// Mitsubishi GX Developer project: may ghep doc 2   PLC: FX1N

PROGRAM MAIN
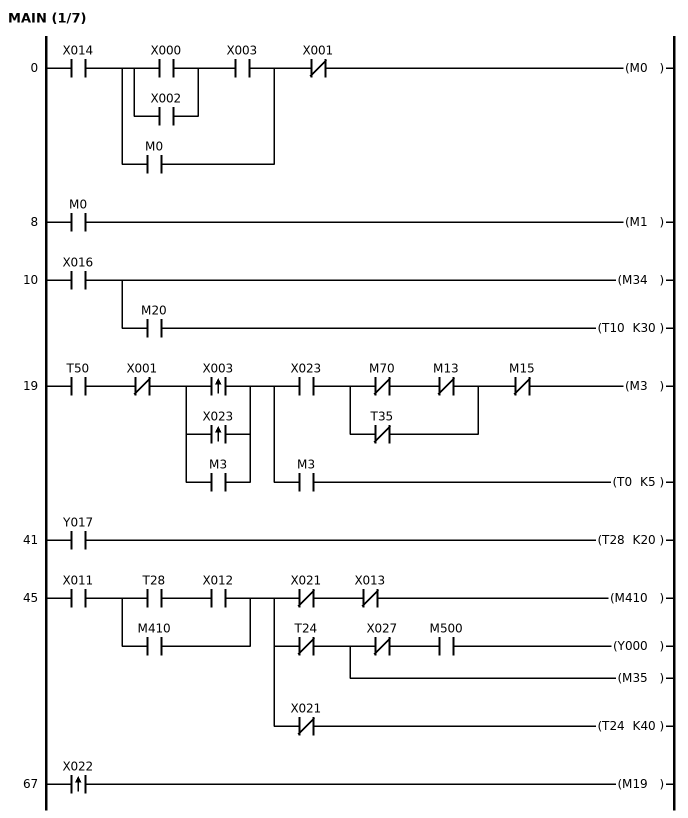
0     LD      X014
      LD      X000
      OR      X002
      AND     X003
      OR      M0
      ANB
      ANI     X001
      OUT     M0
8     LD      M0
      OUT     M1
10    LD      X016
      OUT     M34
      AND     M20
      OUT     T10 K30
19    LD      T50
      ANI     X001
      LDP     X003
      ORP     X023
      OR      M3
      ANB
      MPS
      AND     X023
      LDI     M70
      ANI     M13
      ORI     T35
      ANB
      ANI     M15
      OUT     M3
      MPP
      AND     M3
      OUT     T0 K5
41    LD      Y017
      OUT     T28 K20
45    LD      X011
      LD      T28
      AND     X012
      OR      M410
      ANB
      MPS
      ANI     X021
      ANI     X013
      OUT     M410
      MRD
      ANI     T24
      MPS
      ANI     X027
      AND     M500
      OUT     Y000
      MPP
      OUT     M35
      MPP
      ANI     X021
      OUT     T24 K40
67    LDP     X022
      OUT     M19
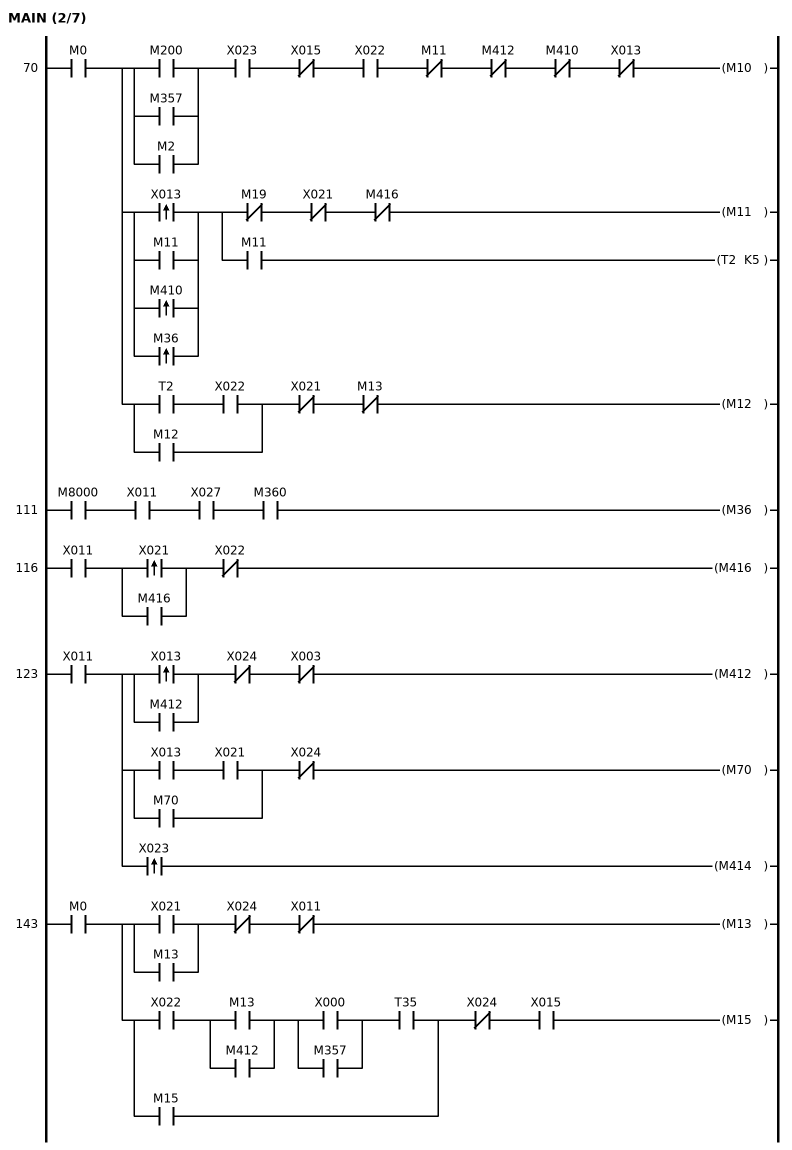
70    LD      M0
      MPS
      LD      M200
      OR      M357
      OR      M2
      ANB
      AND     X023
      ANI     X015
      AND     X022
      ANI     M11
      ANI     M412
      ANI     M410
      ANI     X013
      OUT     M10
      MRD
      LDP     X013
      OR      M11
      ORP     M410
      ORP     M36
      ANB
      MPS
      ANI     M19
      ANI     X021
      ANI     M416
      OUT     M11
      MPP
      AND     M11
      OUT     T2 K5
      MPP
      LD      T2
      AND     X022
      OR      M12
      ANB
      ANI     X021
      ANI     M13
      OUT     M12
111   LD      M8000
      AND     X011
      AND     X027
      AND     M360
      OUT     M36
116   LD      X011
      LDP     X021
      OR      M416
      ANB
      ANI     X022
      OUT     M416
123   LD      X011
      MPS
      LDP     X013
      OR      M412
      ANB
      ANI     X024
      ANI     X003
      OUT     M412
      MRD
      LD      X013
      AND     X021
      OR      M70
      ANB
      ANI     X024
      OUT     M70
      MPP
      ANDP    X023
      OUT     M414
143   LD      M0
      MPS
      LD      X021
      OR      M13
      ANB
      ANI     X024
      ANI     X011
      OUT     M13
      MPP
      LD      X022
      LD      M13
      OR      M412
      ANB
      LD      X000
      OR      M357
      ANB
      AND     T35
      OR      M15
      ANB
      ANI     X024
      AND     X015
      OUT     M15
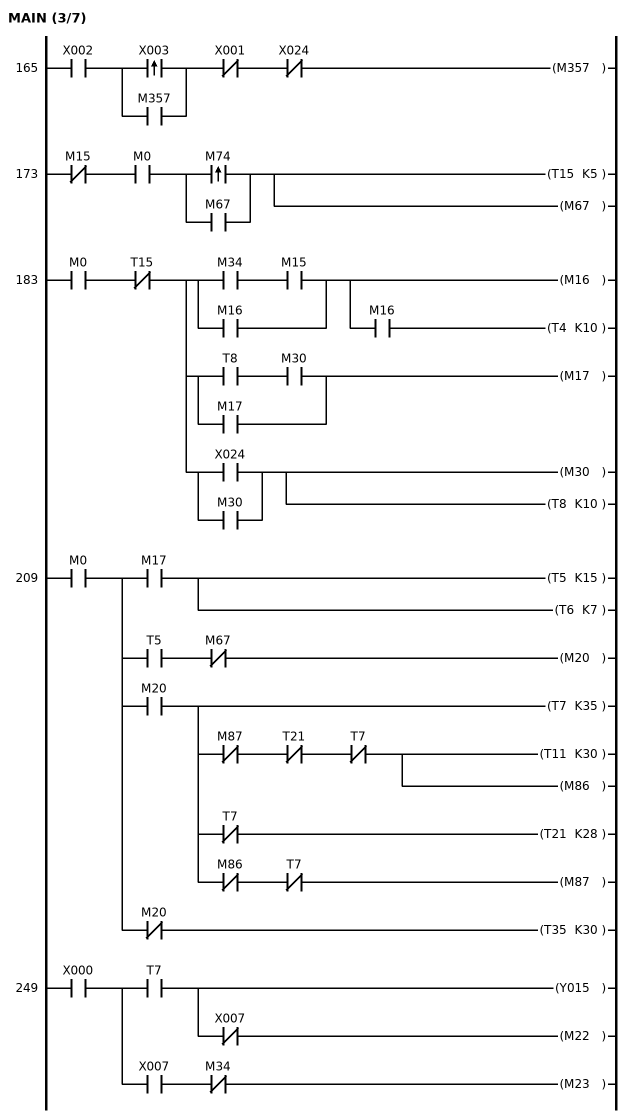
165   LD      X002
      LDP     X003
      OR      M357
      ANB
      ANI     X001
      ANI     X024
      OUT     M357
173   LDI     M15
      AND     M0
      LDP     M74
      OR      M67
      ANB
      OUT     T15 K5
      OUT     M67
183   LD      M0
      ANI     T15
      MPS
      LD      M34
      AND     M15
      OR      M16
      ANB
      OUT     M16
      AND     M16
      OUT     T4 K10
      MRD
      LD      T8
      AND     M30
      OR      M17
      ANB
      OUT     M17
      MPP
      LD      X024
      OR      M30
      ANB
      OUT     M30
      OUT     T8 K10
209   LD      M0
      MPS
      AND     M17
      OUT     T5 K15
      OUT     T6 K7
      MRD
      AND     T5
      ANI     M67
      OUT     M20
      MRD
      AND     M20
      OUT     T7 K35
      MPS
      ANI     M87
      ANI     T21
      ANI     T7
      OUT     T11 K30
      OUT     M86
      MRD
      ANI     T7
      OUT     T21 K28
      MPP
      ANI     M86
      ANI     T7
      OUT     M87
      MPP
      ANI     M20
      OUT     T35 K30
249   LD      X000
      MPS
      AND     T7
      OUT     Y015
      ANI     X007
      OUT     M22
      MPP
      AND     X007
      ANI     M34
      OUT     M23
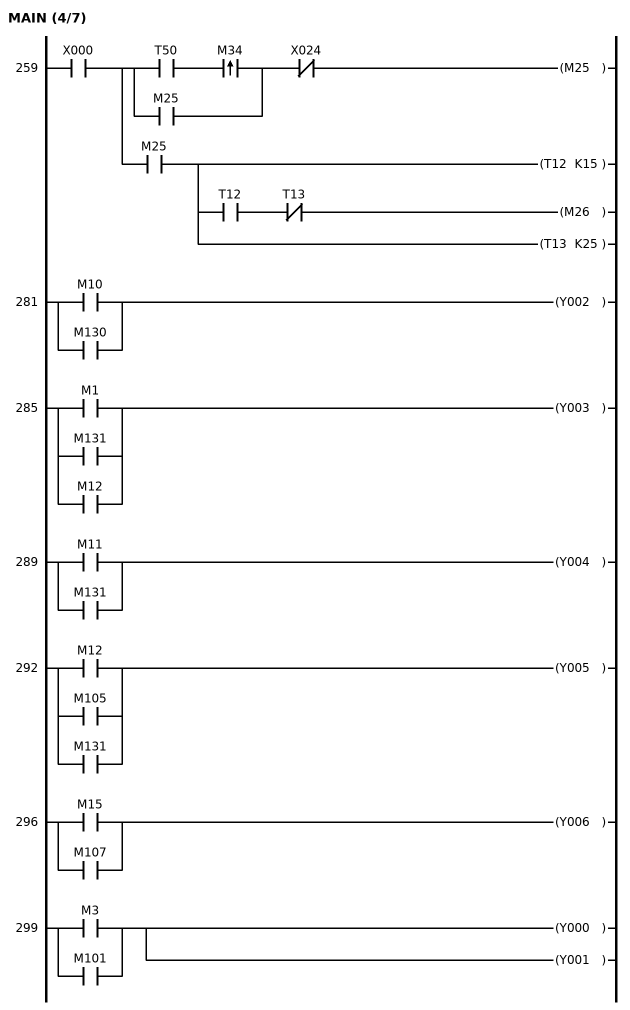
259   LD      X000
      MPS
      LD      T50
      ANDP    M34
      OR      M25
      ANB
      ANI     X024
      OUT     M25
      MPP
      AND     M25
      OUT     T12 K15
      MPS
      AND     T12
      ANI     T13
      OUT     M26
      MPP
      OUT     T13 K25
281   LD      M10
      OR      M130
      OUT     Y002
285   LD      M1
      OR      M131
      OR      M12
      OUT     Y003
289   LD      M11
      OR      M131
      OUT     Y004
292   LD      M12
      OR      M105
      OR      M131
      OUT     Y005
296   LD      M15
      OR      M107
      OUT     Y006
299   LD      M3
      OR      M101
      OUT     Y000
      OUT     Y001
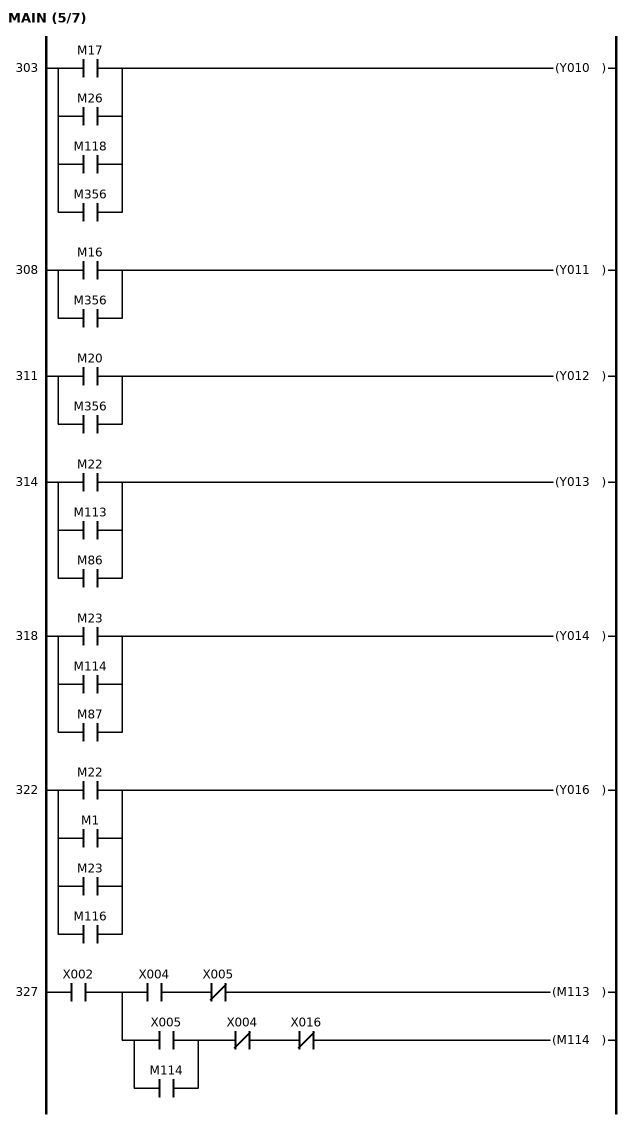
303   LD      M17
      OR      M26
      OR      M118
      OR      M356
      OUT     Y010
308   LD      M16
      OR      M356
      OUT     Y011
311   LD      M20
      OR      M356
      OUT     Y012
314   LD      M22
      OR      M113
      OR      M86
      OUT     Y013
318   LD      M23
      OR      M114
      OR      M87
      OUT     Y014
322   LD      M22
      OR      M1
      OR      M23
      OR      M116
      OUT     Y016
327   LD      X002
      MPS
      AND     X004
      ANI     X005
      OUT     M113
      MPP
      LD      X005
      OR      M114
      ANB
      ANI     X004
      ANI     X016
      OUT     M114
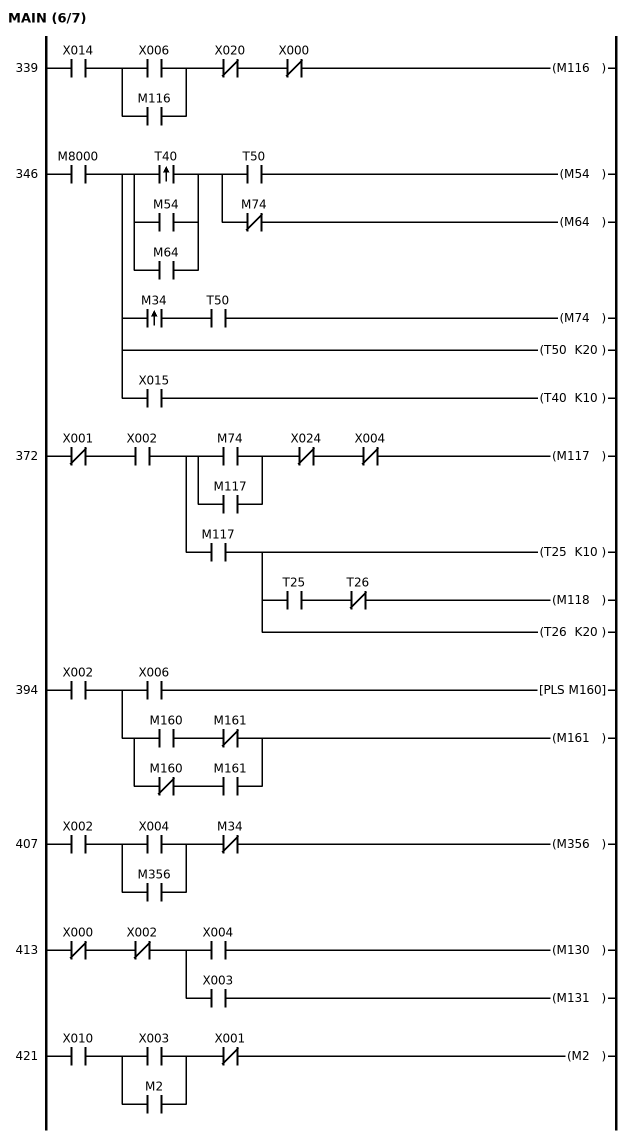
339   LD      X014
      LD      X006
      OR      M116
      ANB
      ANI     X020
      ANI     X000
      OUT     M116
346   LD      M8000
      MPS
      LDP     T40
      OR      M54
      OR      M64
      ANB
      MPS
      AND     T50
      OUT     M54
      MPP
      ANI     M74
      OUT     M64
      MRD
      ANDP    M34
      AND     T50
      OUT     M74
      MPP
      OUT     T50 K20
      AND     X015
      OUT     T40 K10
372   LDI     X001
      AND     X002
      MPS
      LD      M74
      OR      M117
      ANB
      ANI     X024
      ANI     X004
      OUT     M117
      MPP
      AND     M117
      OUT     T25 K10
      MPS
      AND     T25
      ANI     T26
      OUT     M118
      MPP
      OUT     T26 K20
394   LD      X002
      MPS
      AND     X006
      PLS     M160
      MPP
      LD      M160
      ANI     M161
      LDI     M160
      AND     M161
      ORB
      ANB
      OUT     M161
407   LD      X002
      LD      X004
      OR      M356
      ANB
      ANI     M34
      OUT     M356
413   LDI     X000
      ANI     X002
      MPS
      AND     X004
      OUT     M130
      MPP
      AND     X003
      OUT     M131
421   LD      X010
      LD      X003
      OR      M2
      ANB
      ANI     X001
      OUT     M2
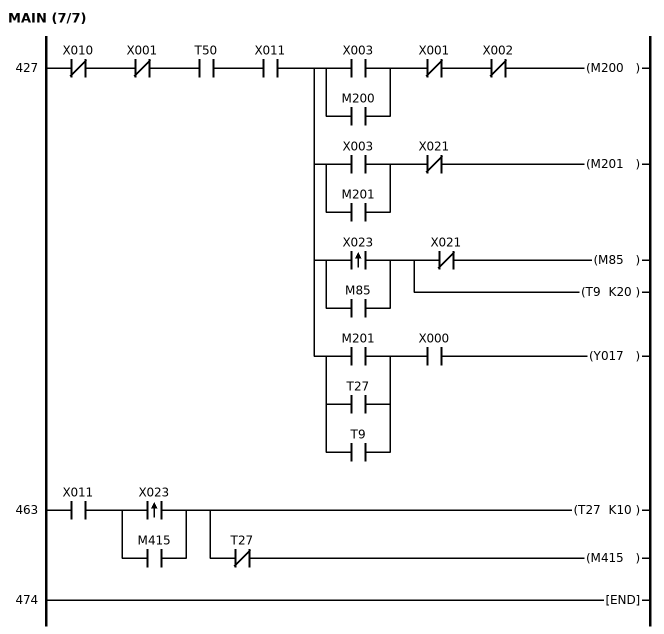
427   LDI     X010
      ANI     X001
      AND     T50
      AND     X011
      MPS
      LD      X003
      OR      M200
      ANB
      ANI     X001
      ANI     X002
      OUT     M200
      MRD
      LD      X003
      OR      M201
      ANB
      ANI     X021
      OUT     M201
      MRD
      LDP     X023
      OR      M85
      ANB
      MPS
      ANI     X021
      OUT     M85
      MPP
      OUT     T9 K20
      MPP
      LD      M201
      OR      T27
      OR      T9
      ANB
      AND     X000
      OUT     Y017
463   LD      X011
      LDP     X023
      OR      M415
      ANB
      OUT     T27 K10
      ANI     T27
      OUT     M415
474   END
END_PROGRAM
